{attribute addProperty BoxType "EP3184-0002-0017"}
{attribute addProperty Id "AI_Standard_ChannelAT %I*ARRAY[0..3] OF AI_Standard_Channel_904746A2128160WcStateAT %I*WcState_98A4DF7520.250InfoDataAT %I*InfoData_BC63D37F80100"}
{attribute addProperty CRC "1712706657"}
{attribute addProperty SizeInBites "210"}
{attribute addProperty SizeInBytes "26.25"}
TYPE EP3184_6082EBFD :
STRUCT
	{attribute addProperty Name "AI_Standard_Channel"}
	AI_Standard_Channel : ARRAY[0..3] OF AI_Standard_Channel_904746A2;
	{attribute addProperty Name "WcState"}
	WcState : WcState_98A4DF75;
	{attribute addProperty Name "InfoData"}
	InfoData : InfoData_BC63D37F;
END_STRUCT
END_TYPE

(* stored: Version 1.2.0.0, ProductVersion 3.1.4024.9
   DUT EP3184_6082EBFD: Id {f2e4dda3-0e5c-4e2c-926a-0549d03644e4} *)
